FUNCTION_BLOCK FB_Ethercat EXTENDS FB_Component
VAR_INPUT
END_VAR
VAR_OUTPUT
END_VAR
VAR
	AmsNetID					AT%I*:AmsNetID;	
	fbGetSlaveStates:			FB_EcGetAllSlaveStates;
	aSlaveState:				ARRAY [0..EC_MAX_SLAVES] OF ST_EcSlaveState;
END_VAR

SUPER^();

METHOD PROTECTED M_Execute : BOOL (* Return*)
// 
// fbGetSlaveStates(sNetId:= AmsNetID, ADR(a)

M_Execute:= TRUE;
END_METHOD

METHOD PROTECTED M_Starting : BOOL (* Return state complete*)
fbGetSlaveCount.sNetId:= AmsNetID;
fbGetSlaveCount.bExecute:= TRUE;

M_Starting:= TRUE;
END_METHOD

END_FUNCTION_BLOCK

(* stored: Version 1.1.0.1
   POU FB_Ethercat: Id {62ca7924-6364-0c5a-06c4-f002022b97f1}, SpecialFunc None
   Method M_Execute: Id {4e92595d-432e-0baf-3e87-fcbfb8b200aa}
   Method M_Starting: Id {01edd329-ad62-031a-014c-c40cc08b18f9} *)
